Staubli VAL3: robotMove.pgx

public program robotMove(num& x_nHostRosFlag, num& x_nRobotFlag, num& x_nForceFlag, jointRx& x_jRobotMove)
begin

  //This program is used for realtime robot control, and it should be called every 4ms(standard robot loop time).
  //It will move the robot to the given goal position based on the current judging condition(robot condition and
  //contact force) in every 4ms. And the program will keep the current judging condition interface reserved for
  //future function expansion.

  //Judge the current host ROS command, robot status and contact force and then decide whether the loop will begin.
  while (x_nHostRosFlag==1 and x_nRobotFlag==1 and x_nForceFlag==1)

    //Send the joint command for the next 4ms, and returns true if command accepted, false if refuesed.(movejSync
    //instruction not started or already completed.)
    if(!$movejSync(x_jRobotMove))
      popUpMsg("The joint motion command refused and robot will stop.")
      return
    endIf

    //Force the sequencing to the next task by using the "delay(0.0)" instruction explicitly.
    delay(0.0)

  endWhile

  //End the Sychronous Movej procedural motion mode and stop the robot.
  $movejSyncEnd()
  stopMove()

end
